Staubli VAL3: getErrorMessage.pgx

public program getErrorMessage(string& x_sMessage[])
begin

  // This programs returns a clear text about the last error code

  //

  // Input Param

  // None

  //

  // Output Param

  //  x_sMessage    : Error message

  //

  //Created 21/12/05                              C.CURRIVAND

  //--------------------------------------------------------------

  x_sMessage=sErrorMessage

end
